// Mitsubishi GX Works2 project: LAB3TASK3   PLC: FX1S

PROGRAM MAIN
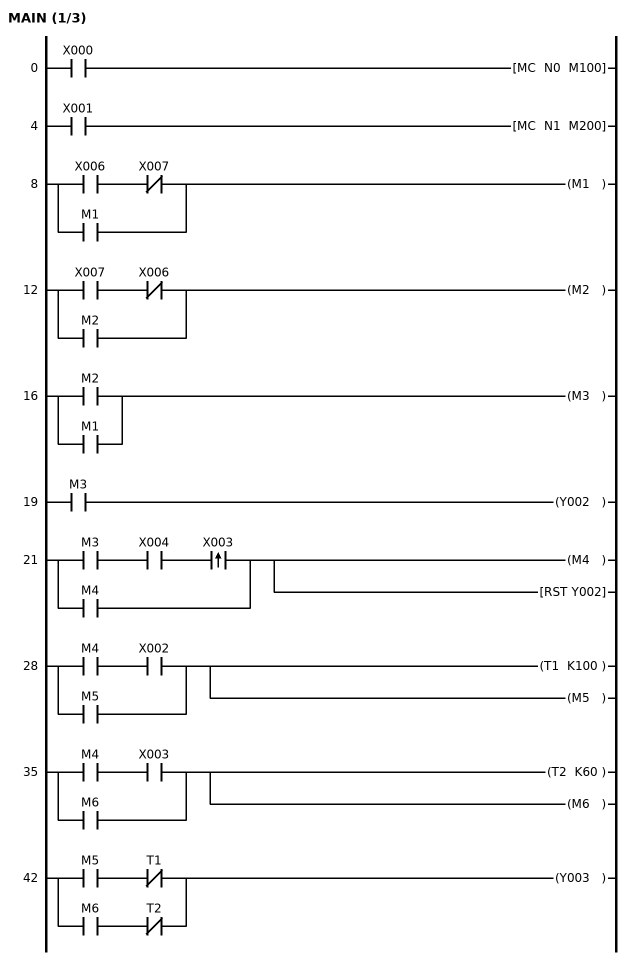
0     LD      X000
      MC      N0 M100
4     LD      X001
      MC      N1 M200
8     LD      X006
      ANI     X007
      OR      M1
      OUT     M1
12    LD      X007
      ANI     X006
      OR      M2
      OUT     M2
16    LD      M2
      OR      M1
      OUT     M3
19    LD      M3
      OUT     Y002
21    LD      M3
      AND     X004
      ANDP    X003
      OR      M4
      OUT     M4
      RST     Y002
28    LD      M4
      AND     X002
      OR      M5
      OUT     T1 K100
      OUT     M5
35    LD      M4
      AND     X003
      OR      M6
      OUT     T2 K60
      OUT     M6
42    LD      M5
      ANI     T1
      LD      M6
      ANI     T2
      ORB
      OUT     Y003
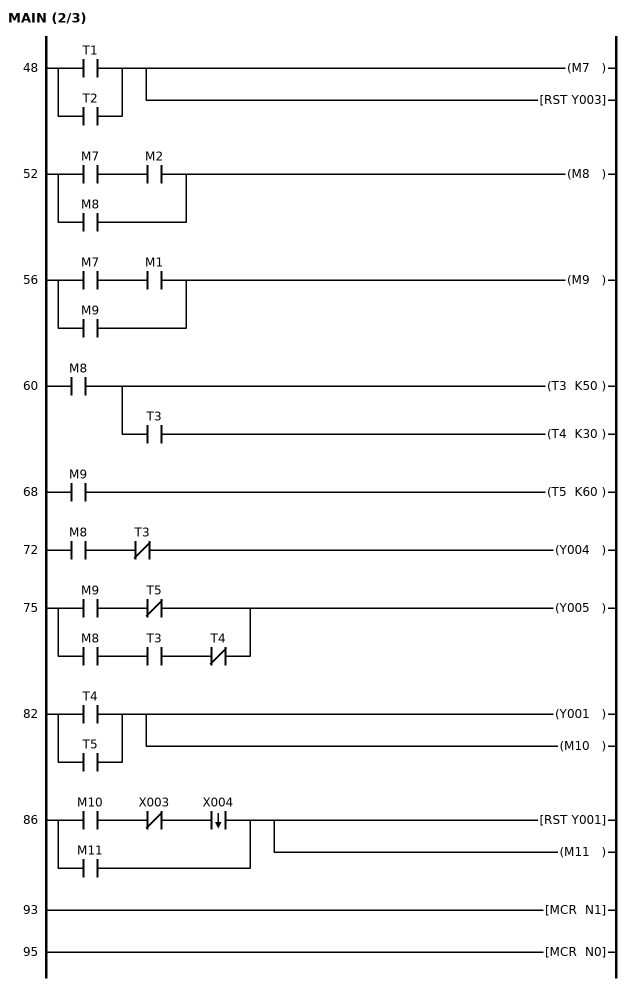
48    LD      T1
      OR      T2
      OUT     M7
      RST     Y003
52    LD      M7
      AND     M2
      OR      M8
      OUT     M8
56    LD      M7
      AND     M1
      OR      M9
      OUT     M9
60    LD      M8
      OUT     T3 K50
      AND     T3
      OUT     T4 K30
68    LD      M9
      OUT     T5 K60
72    LD      M8
      ANI     T3
      OUT     Y004
75    LD      M9
      ANI     T5
      LD      M8
      AND     T3
      ANI     T4
      ORB
      OUT     Y005
82    LD      T4
      OR      T5
      OUT     Y001
      OUT     M10
86    LD      M10
      ANI     X003
      ANDF    X004
      OR      M11
      RST     Y001
      OUT     M11
93    MCR     N1
95    MCR     N0
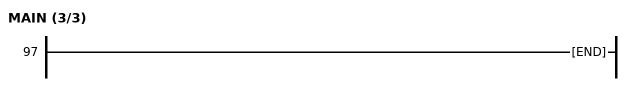
97    END
END_PROGRAM
